Yaskawa INFORM job: OUTPUT.JBI

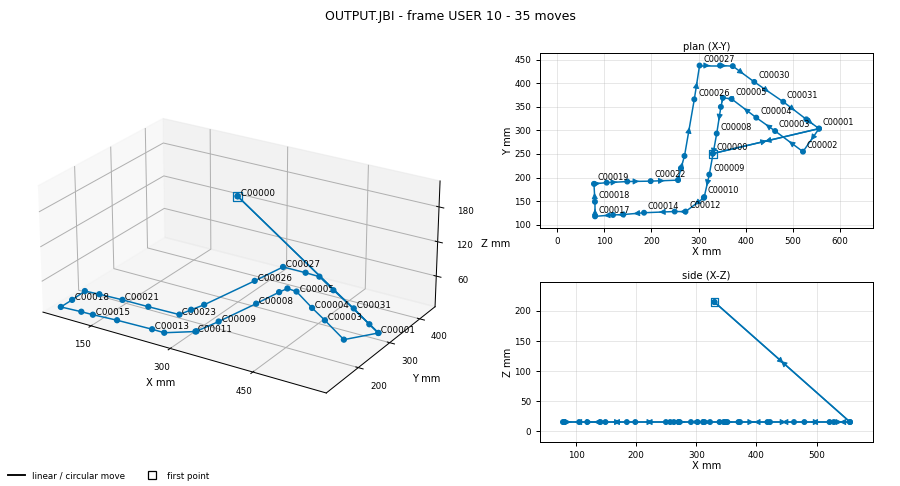
[picture p0: tool path of OUTPUT.JBI in frame USER 10, 35 of 35 moves have a stored position in this frame; points joined in program order, loops and branches not executed]
/JOB
//NAME MOV_IMG
//POS
///NPOS 35,0,0,0,0,0
///TOOL 1
///USER 10
///POSTYPE USER
///RECTAN
///RCONF 0,0,0,0,0,0,0,0
C00000=330.163,250.900,214.789,179.5565,0.1831,0.3047
C00001=555.742,303.856,15.173,179.5565,0.1831,0.3047
C00002=521.653,254.957,15.173,179.5565,0.1831,0.3047
C00003=462.522,298.731,15.173,179.5565,0.1831,0.3047
C00004=422.541,327.131,15.173,179.5565,0.1831,0.3047
C00005=370.144,366.848,15.173,179.5565,0.1831,0.3047
C00006=351.626,369.197,15.173,179.5565,0.1831,0.3047
C00007=347.418,349.979,15.173,179.5565,0.1831,0.3047
C00008=338.580,293.393,15.173,179.5565,0.1831,0.3047
C00009=322.797,206.272,15.173,179.5565,0.1831,0.3047
C00010=312.066,158.654,15.173,179.5565,0.1831,0.3047
C00011=311.224,156.946,15.173,179.5565,0.1831,0.3047
C00012=272.295,127.692,15.173,179.5565,0.1831,0.3047
C00013=249.358,127.906,15.173,179.5565,0.1831,0.3047
C00014=184.335,125.343,15.173,179.5565,0.1831,0.3047
C00015=140.356,121.500,15.173,179.5565,0.1831,0.3047
C00016=118.471,120.646,15.173,179.5565,0.1831,0.3047
C00017=80.384,117.656,15.173,179.5565,0.1831,0.3047
C00018=80.173,148.618,15.173,179.5565,0.1831,0.3047
C00019=78.069,186.627,15.173,179.5565,0.1831,0.3047
C00020=105.004,189.189,15.173,179.5565,0.1831,0.3047
C00021=148.773,191.538,15.173,179.5565,0.1831,0.3047
C00022=198.434,192.392,15.173,179.5565,0.1831,0.3047
C00023=256.512,194.528,15.173,179.5565,0.1831,0.3047
C00024=262.615,219.297,15.173,179.5565,0.1831,0.3047
C00025=270.190,245.775,15.173,179.5565,0.1831,0.3047
C00026=291.023,365.994,15.173,179.5565,0.1831,0.3047
C00027=302.175,437.740,15.173,179.5565,0.1831,0.3047
C00028=345.524,437.740,15.173,179.5565,0.1831,0.3047
C00029=372.669,436.459,15.173,179.5565,0.1831,0.3047
C00030=418.332,402.935,15.173,179.5565,0.1831,0.3047
C00031=479.777,360.869,15.173,179.5565,0.1831,0.3047
C00032=528.807,323.501,15.173,179.5565,0.1831,0.3047
C00033=555.742,303.856,15.173,179.5565,0.1831,0.3047
C00034=330.163,250.900,214.789,179.5565,0.1831,0.3047
//INST
///DATE 2017/14/12 09:00
///ATTR SC,RW,RJ
///GROUP1 RB1
NOP
MOVL C00000 V=41.7
MOVL C00001 V=41.7
MOVL C00002 V=41.7
MOVL C00003 V=41.7
MOVL C00004 V=41.7
MOVL C00005 V=41.7
MOVL C00006 V=41.7
MOVL C00007 V=41.7
MOVL C00008 V=41.7
MOVL C00009 V=41.7
MOVL C00010 V=41.7
MOVL C00011 V=41.7
MOVL C00012 V=41.7
MOVL C00013 V=41.7
MOVL C00014 V=41.7
MOVL C00015 V=41.7
MOVL C00016 V=41.7
MOVL C00017 V=41.7
MOVL C00018 V=41.7
MOVL C00019 V=41.7
MOVL C00020 V=41.7
MOVL C00021 V=41.7
MOVL C00022 V=41.7
MOVL C00023 V=41.7
MOVL C00024 V=41.7
MOVL C00025 V=41.7
MOVL C00026 V=41.7
MOVL C00027 V=41.7
MOVL C00028 V=41.7
MOVL C00029 V=41.7
MOVL C00030 V=41.7
MOVL C00031 V=41.7
MOVL C00032 V=41.7
MOVL C00033 V=41.7
MOVL C00034 V=41.7
END
